FUNCTION_BLOCK SludgeBufferSensors_2 (* Composite Function Block Type *)
  (* Standard: 61499-2 *)
  (* Version 1.0, 9/30/2026, Claude/Hidryco, Schneider Electric, Rev1 - 49FT0004 exposto em PV3..PV5 para as fases de descarga *)
  PACKAGE SE.Nereda;
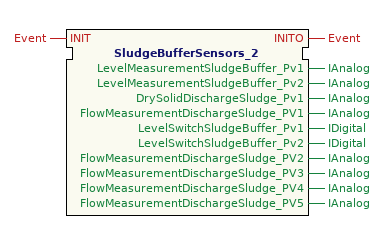
  EVENT_INPUT
    INIT;
  END_EVENT
  EVENT_OUTPUT
    INITO;
  END_EVENT
  PLUGS
    LevelMeasurementSludgeBuffer_Pv1 : IAnalog; (* Process value and status interface adapter *)
    LevelMeasurementSludgeBuffer_Pv2 : IAnalog; (* Process value and status interface adapter *)
    DrySolidDischargeSludge_Pv1 : IAnalog; (* Process value and status interface adapter *)
    FlowMeasurementDischargeSludge_PV1 : IAnalog; (* Process value and status interface adapter *)
    LevelSwitchSludgeBuffer_Pv1 : IDigital; (* Process value interface adapter *)
    LevelSwitchSludgeBuffer_Pv2 : IDigital; (* Process value interface adapter *)
    FlowMeasurementDischargeSludge_PV2 : IAnalog; (* Process value and status interface adapter *)
    FlowMeasurementDischargeSludge_PV3 : IAnalog; (* 49FT0004 - vazao descarga SB *)
    FlowMeasurementDischargeSludge_PV4 : IAnalog; (* 49FT0004 - vazao descarga SB *)
    FlowMeasurementDischargeSludge_PV5 : IAnalog; (* 49FT0004 - vazao descarga SB *)
  END_PLUGS
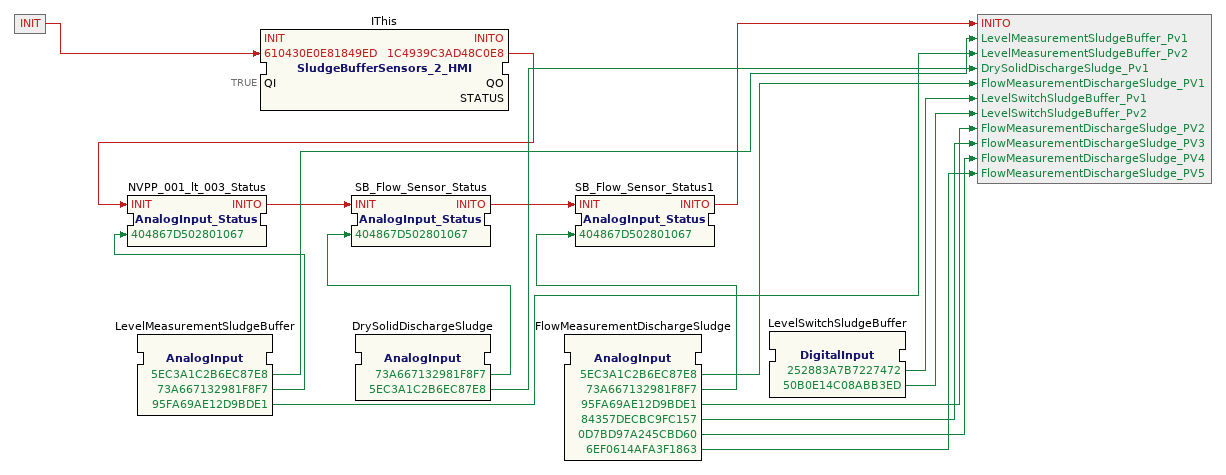
  (* 01 - FUNCTIONNAL INPUT INTERFACE *)
  (* 00 - INITIALIZATION *)
  (* 06 - HMI INTERFACE *)
  (* 02 - FUNCTIONNAL OUTPUT INTERFACE *)
  (* 03 - FIELD INTERFACE *)
  (* Level measurement sludge buffer *)
  (* Dry Solid discharge sludge *)
  (* 05 - LOGIC *)
  (* Actuators Status *)
  (* Flow Measurement discharge sludge *)
  (* Level Switch sludge buffer *)
  FBS
    IThis : SludgeBufferSensors_2_HMI(QI := TRUE);
    LevelMeasurementSludgeBuffer : AnalogInput;
    DrySolidDischargeSludge : AnalogInput;
    NVPP_001_lt_003_Status : AnalogInput_Status;
    SB_Flow_Sensor_Status : AnalogInput_Status;
    FlowMeasurementDischargeSludge : AnalogInput;
    LevelSwitchSludgeBuffer : DigitalInput;
    SB_Flow_Sensor_Status1 : AnalogInput_Status;
  END_FBS
  EVENT_CONNECTIONS
    INIT TO IThis.610430E0E81849ED;
    NVPP_001_lt_003_Status.INITO TO SB_Flow_Sensor_Status.INIT;
    IThis.1C4939C3AD48C0E8 TO NVPP_001_lt_003_Status.INIT;
    SB_Flow_Sensor_Status1.INITO TO INITO;
    SB_Flow_Sensor_Status.INITO TO SB_Flow_Sensor_Status1.INIT;
  END_CONNECTIONS
  ADAPTER_CONNECTIONS
    LevelMeasurementSludgeBuffer.5EC3A1C2B6EC87E8 TO LevelMeasurementSludgeBuffer_Pv1;
    LevelMeasurementSludgeBuffer.73A667132981F8F7 TO NVPP_001_lt_003_Status.404867D502801067;
    DrySolidDischargeSludge.73A667132981F8F7 TO SB_Flow_Sensor_Status.404867D502801067;
    LevelSwitchSludgeBuffer.252883A7B7227472 TO LevelSwitchSludgeBuffer_Pv1;
    FlowMeasurementDischargeSludge.5EC3A1C2B6EC87E8 TO FlowMeasurementDischargeSludge_PV1;
    FlowMeasurementDischargeSludge.73A667132981F8F7 TO SB_Flow_Sensor_Status1.404867D502801067;
    DrySolidDischargeSludge.5EC3A1C2B6EC87E8 TO DrySolidDischargeSludge_Pv1;
    LevelMeasurementSludgeBuffer.95FA69AE12D9BDE1 TO LevelMeasurementSludgeBuffer_Pv2;
    LevelSwitchSludgeBuffer.50B0E14C08ABB3ED TO LevelSwitchSludgeBuffer_Pv2;
    FlowMeasurementDischargeSludge.95FA69AE12D9BDE1 TO FlowMeasurementDischargeSludge_PV2;
    FlowMeasurementDischargeSludge.84357DECBC9FC157 TO FlowMeasurementDischargeSludge_PV3;
    FlowMeasurementDischargeSludge.0D7BD97A245CBD60 TO FlowMeasurementDischargeSludge_PV4;
    FlowMeasurementDischargeSludge.6EF0614AFA3F1863 TO FlowMeasurementDischargeSludge_PV5;
  END_CONNECTIONS
END_FUNCTION_BLOCK
